// SIMATIC S7-200 project (STEP 7-Micro/WIN), CPU 221 REL 01.10

ORGANIZATION_BLOCK PRINCIPAL:OB1
TITLE=COMENTARIOS DEL PROGRAMA
BEGIN
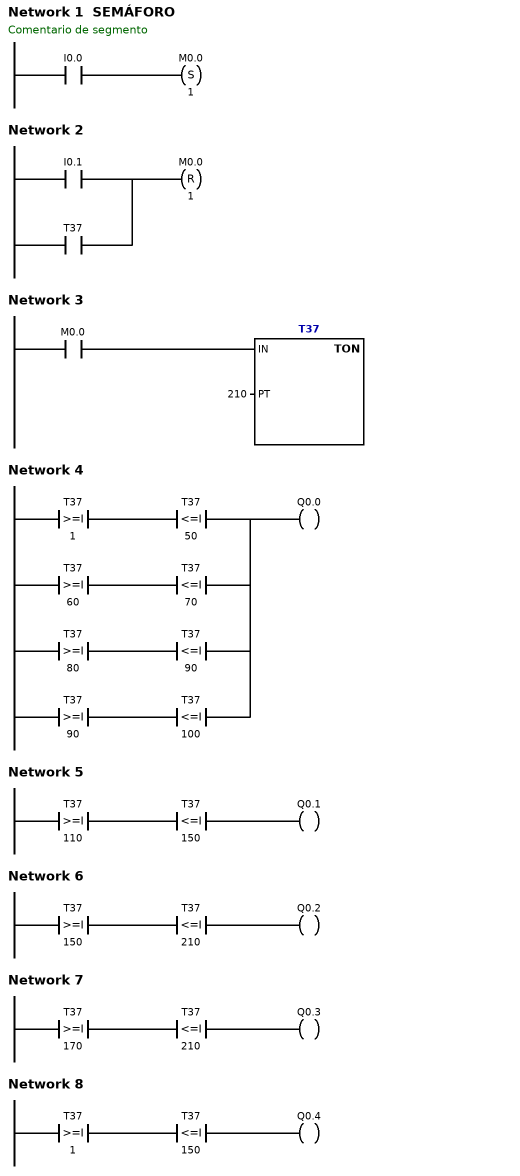
Network 1 // SEMÁFORO
// Comentario de segmento
LD     I0.0
S      M0.0, 1
Network 2
LD     I0.1
O      T37
R      M0.0, 1
Network 3
LD     M0.0
TON    T37, 210
Network 4
LDW>=  T37, 1
AW<=   T37, 50
LDW>=  T37, 60
AW<=   T37, 70
OLD
LDW>=  T37, 80
AW<=   T37, 90
OLD
LDW>=  T37, 90
AW<=   T37, 100
OLD
=      Q0.0
Network 5
LDW>=  T37, 110
AW<=   T37, 150
=      Q0.1
Network 6
LDW>=  T37, 150
AW<=   T37, 210
=      Q0.2
Network 7
LDW>=  T37, 170
AW<=   T37, 210
=      Q0.3
Network 8
LDW>=  T37, 1
AW<=   T37, 150
=      Q0.4
END_ORGANIZATION_BLOCK
